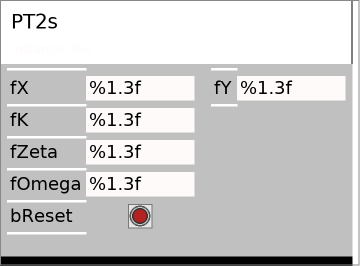
VISUALIZATION RET_VISU_PT2s  // 360x266
VAR_INPUT
   {attribute 'parameterstringof' := 'm_Input_FB'}
   m_Input_INST_Str : STRING;
END_VAR
VAR_IN_OUT
   m_Input_FB : PT2s;
END_VAR
    RoundedRectangle (0,0 352x81)
    RoundedRectangle (0,226 352x40)
    Rectangle (0,64 352x192)
    PushSwitch (128,204 24x24), variable: m_Input_FB.bReset, behaviour: TOGGLE, style: Switch-PushSwitch-Red
    Rectangle (8,8 352x27), "PT2s"
    Rectangle (8,35 352x27), "Instance: %s", text variable: m_Input_INST_Str
    Rectangle (7,68 79x2)
    Rectangle (86,76 108x24), "%1.3f", text variable: m_Input_FB.fX
        OnMouseClick: write the text variable via Default
    Rectangle (7,76 79x24), "fX"
    Rectangle (7,104 79x2)
    Rectangle (86,108 108x24), "%1.3f", text variable: m_Input_FB.fK
        OnMouseClick: write the text variable via Default
    Rectangle (7,108 79x24), "fK"
    Rectangle (7,136 79x2)
    Rectangle (86,140 108x24), "%1.3f", text variable: m_Input_FB.fZeta
        OnMouseClick: write the text variable via Default
    Rectangle (7,140 79x24), "fZeta"
    Rectangle (7,168 79x2)
    Rectangle (86,172 108x24), "%1.3f", text variable: m_Input_FB.fOmega
        OnMouseClick: write the text variable via Default
    Rectangle (7,172 79x24), "fOmega"
    Rectangle (7,200 79x2)
    Rectangle (7,204 79x24), "bReset"
    Rectangle (7,232 79x2)
    Rectangle (211,68 26x2)
    Rectangle (237,76 108x24), "%1.3f", text variable: m_Input_FB.fY
    Rectangle (211,76 26x24), "fY"
    Rectangle (211,104 26x2)
END_VISUALIZATION

(* stored: Version 1.1.0.1, ProductVersion 3.1.4024.12
   Visu RET_VISU_PT2s: Id {18a54949-e0fe-48a4-a96e-14af1191f650} *)
